// TwinCAT 3 PLC project _00_Strategy
// ProgramVersion: 3.1.4023.0
// libraries:
//   Tc2_Standard, * (Beckhoff Automation GmbH)
//   Tc2_System, * (Beckhoff Automation GmbH)
//   Tc3_Module, * (Beckhoff Automation GmbH)
// project tree:
//   Helpers/ C_TO_F.TcPOU (not stored), RES_PT.TcPOU (not stored), TEMP_PT.TcPOU (not stored)
//   / MAIN.TcPOU, PlcTask.TcTTO (not stored)
//   Strategy Pattern/General/Temperature sensor/ tempSensor_PT100.TcPOU (not stored), tempSensor_PT1000.TcPOU, tempSensor.TcPOU (not stored)
//   Strategy Pattern/Interfaces/ ITempSensor.TcIO
//   Strategy Pattern/Motors/ motor.TcPOU (not stored)
//   Strategy Pattern/ P_Strategy.TcPOU
// real-time tasks:
//   TASK PlcTask: cycle T#10ms, priority 20, ADS port 350

// ---- Strategy Pattern/Interfaces/ITempSensor.TcIO
INTERFACE ITempSensor

PROPERTY tempDegreesC : real
GET
END_GET
END_PROPERTY

PROPERTY tempDegreesF : real
GET
END_GET
END_PROPERTY

END_INTERFACE

// ---- MAIN.TcPOU
PROGRAM MAIN
VAR
END_VAR

P_Strategy();

END_PROGRAM

// ---- Strategy Pattern/P_Strategy.TcPOU
PROGRAM P_Strategy
VAR
	// instantiations of concrete classes 
	sensor1_1		: tempSensor_PT100;
	sensor1_2		: tempSensor_PT1000;
	motor1			: motor(tempSensor := sensor1_1);
	sensor2			: tempSensor_PT1000;
	motor2			: motor(sensor2);
	
	// Change the sensor during runtime
	useSensor2		: BOOL;
	
	// Debug
	motor1_Temp		: REAL;
	motor2_Temp		: REAL;	
END_VAR
(*
Strategy allows one of a family of algorithms to be selected on-the-fly at runtime.
https://en.wikipedia.org/wiki/Strategy_pattern
*)

// Motors
motor1.cyclicCall();	
motor2.cyclicCall();	

// Change the temperature sensor of motor 1 during runtime
IF useSensor2		THEN
	motor1.changeTempSensor := sensor1_2;
ELSE
	motor1.changeTempSensor := sensor1_1;	
END_IF

sensor1_1.DEBUG_setRawValue := 110;
sensor1_2.DEBUG_setRawValue := 1010;
sensor2.DEBUG_setRawValue := 1010;

// Motor temperature feedback
motor1_Temp := motor1.motorTemperature;
motor2_Temp := motor2.motorTemperature;

END_PROGRAM

// ---- Strategy Pattern/General/Temperature sensor/tempSensor_PT1000.TcPOU
{attribute 'no_explicit_call' := 'This is a CLASS and should be accessed using methods or properties'}
FUNCTION_BLOCK tempSensor_PT1000 EXTENDS tempSensor
(*~
<docu>
	<summary>
			Implementation of a PT1000 Temperature sensor class based on the base class tempSensor

			Usage:
			degreesC / degreesF return the Celcius / Fahrenheit value determined by the appropriate formula 		
	</summary>				
</docu>	
~*)

(*  
	Principally a CLASS should be accessed using methods or properties
	Good practice is not put code here, or call the class directly 
	Or maybe just a call to a method calling the cyclic code 
*)

PROPERTY tempDegreesC : REAL
GET
tempDegreesC := TEMP_PT(
			Res	:= TO_REAL(rawValue), 
			R0	:= 1000.0
			);
END_GET
END_PROPERTY

END_FUNCTION_BLOCK
